Fanuc KAREL source: kb00044.KL

-- PROVISIONAL review KL for V770-1; original PC SHA256 61ba038b332552c4c1a77d3bb7f9baaf60402503ed7dbca730d3fca73d722674
-- Incomplete behavior may be omitted. Consult companion uncertainty JSON. Do not deploy.
PROGRAM KB00044
%NOLOCKGROUP
BEGIN
  -- UNRESOLVED_PC offsets 5-14; opcodes 3F,75
  -- UNRESOLVED_PC offsets 19-28; opcodes 3F,75
  -- UNRESOLVED_PC offsets 33-40; opcodes 9D,23
  -- UNRESOLVED_PC offsets 45-52; opcodes 9D,23
  -- UNRESOLVED_PC offsets 57-64; opcodes 9D,23
  -- UNRESOLVED_PC offsets 69-113; opcodes 27,22,2A,22,2A,22,22,22,22,31
  -- UNRESOLVED_PC offsets 118-122; opcodes 7F
END KB00044
